{attribute 'qualified_only'}
{attribute 'strict'}
TYPE
    E_FeedInToWareHouse_PlaceArea :
    (
        Undefined := 0,
        WareHouseA := 1,
        WareHouseB := 2,
		PullOutInner := 3,  // PullOutConveyor I3_Slide (左側,面對操作員 / 機台內側)
        PullOutOuter := 4   // PullOutConveyor I4_Slide (右側,面對操作員 / 機台外側)
    )UINT;
END_TYPE

(* stored: Version 1.1.0.1, ProductVersion 3.1.4024.13
   DUT E_FeedInToWareHouse_PlaceArea: Id {a1b2c3d4-1111-4aaa-b111-111111111111} *)
